Omron Sysmac Studio project ScaleTrans_TimeToSec_Ornegi (Sysmac Studio 1.65.0.64007, StandardProject)

# Controller new_Controller_0: NX1P2-1040DT1 version 1.69
Task PrimaryTask (priority 4, period or condition 2000): Program0

VAR_GLOBAL RETAIN
    E_Start_Butonu : BOOL;  (* published *)
    E_Stop_Butonu : BOOL;  (* published *)
END_VAR
VAR_GLOBAL
    OUT_KirmiziLamba : BOOL;  (* published *)
    E_Sari_Lamba_Kalan_Sure : REAL;  (* published *)
    OUT_SariLamba : BOOL;  (* published *)
    OUT_YesilLamba : BOOL;  (* published *)
    E_Yesil_Lamba_Kalan_Sure : REAL;  (* published *)
    E_Kirmizi_Lamba_Kalan_Suree : REAL;
END_VAR

PROGRAM Program0
VAR
    Sistem_Start : BOOL;
    Ton_Dongu : TON;
    Ton_ElapsedTime : TIME;
    REAL_ElapsedTime : REAL;
    LINT_ElapsedTime : LINT;
END_VAR
VAR_EXTERNAL
    E_Start_Butonu : BOOL;
    E_Stop_Butonu : BOOL;
    OUT_KirmiziLamba : BOOL;
    E_Sari_Lamba_Kalan_Sure : REAL;
    OUT_SariLamba : BOOL;
    OUT_YesilLamba : BOOL;
    E_Yesil_Lamba_Kalan_Sure : REAL;
    E_Kirmizi_Lamba_Kalan_Suree : REAL;
END_VAR
VAR
    _p1 : BOOL;
    _p2 : BOOL;
    _p3 : BOOL;
END_VAR

(* Section TrafficLamp: ladder, written here as Structured Text *)

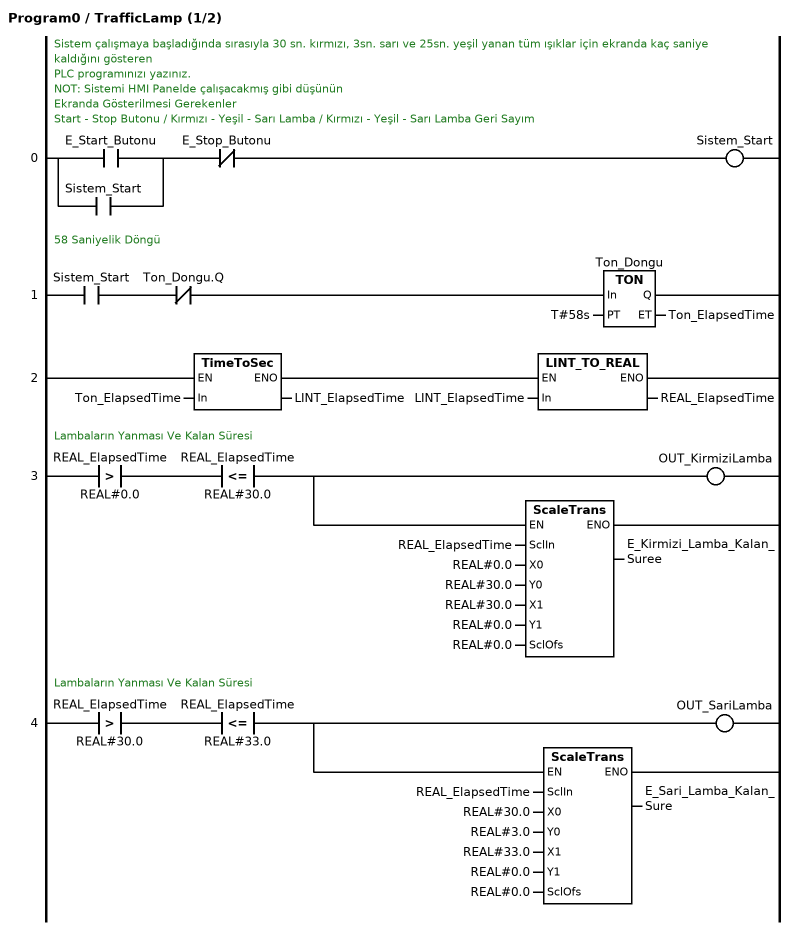
(* Rung 0: Sistem çalışmaya başladığında sırasıyla 30 sn. kırmızı, 3sn. sarı ve 25sn. yeşil yanan tüm ışıklar için ekranda kaç saniye kaldığını gösteren / PLC programınızı yazınız. / NOT: Sistemi HMI Panelde çalışacakmış gibi düşünün / Ekranda Gösterilmesi Gerekenler / Start - Stop Butonu / Kırmızı - Yeşil - Sarı Lamba / Kırmızı - Yeşil - Sarı Lamba Geri Sayım *)
Sistem_Start := (E_Start_Butonu OR Sistem_Start) AND NOT E_Stop_Butonu;
(* Rung 1: 58 Saniyelik Döngü *)
Ton_Dongu(In := Sistem_Start AND NOT Ton_Dongu.Q, PT := T#58s, ET => Ton_ElapsedTime);
(* Rung 2 *)
LINT_ElapsedTime := TimeToSec(In := Ton_ElapsedTime);
REAL_ElapsedTime := LINT_TO_REAL(In := LINT_ElapsedTime);
(* Rung 3: Lambaların Yanması Ve Kalan Süresi *)
_p1 := (REAL_ElapsedTime > REAL#0.0) AND (REAL_ElapsedTime <= REAL#30.0);
OUT_KirmiziLamba := _p1;
IF _p1 THEN
    E_Kirmizi_Lamba_Kalan_Suree := ScaleTrans(SclIn := REAL_ElapsedTime, X0 := REAL#0.0, Y0 := REAL#30.0, X1 := REAL#30.0, Y1 := REAL#0.0, SclOfs := REAL#0.0);
END_IF;
(* Rung 4: Lambaların Yanması Ve Kalan Süresi *)
_p2 := (REAL_ElapsedTime > REAL#30.0) AND (REAL_ElapsedTime <= REAL#33.0);
OUT_SariLamba := _p2;
IF _p2 THEN
    E_Sari_Lamba_Kalan_Sure := ScaleTrans(SclIn := REAL_ElapsedTime, X0 := REAL#30.0, Y0 := REAL#3.0, X1 := REAL#33.0, Y1 := REAL#0.0, SclOfs := REAL#0.0);
END_IF;

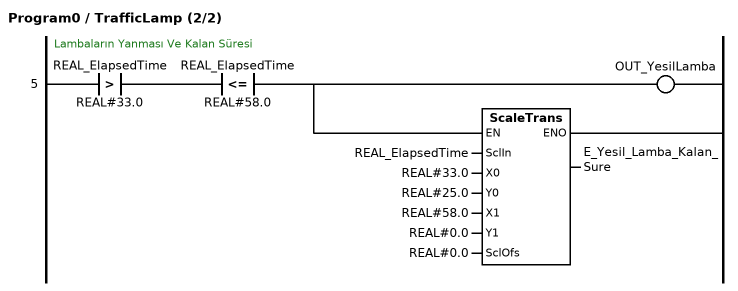
(* Rung 5: Lambaların Yanması Ve Kalan Süresi *)
_p3 := (REAL_ElapsedTime > REAL#33.0) AND (REAL_ElapsedTime <= REAL#58.0);
OUT_YesilLamba := _p3;
IF _p3 THEN
    E_Yesil_Lamba_Kalan_Sure := ScaleTrans(SclIn := REAL_ElapsedTime, X0 := REAL#33.0, Y0 := REAL#25.0, X1 := REAL#58.0, Y1 := REAL#0.0, SclOfs := REAL#0.0);
END_IF;
END_PROGRAM